TYPE ST_TrackStatus :
STRUCT
	MergePermIntlk : ARRAY[GC.MIN_MERGE_PERMINTLK..GC.MAX_MERGE_PERMINTLK] OF BOOL;
END_STRUCT
END_TYPE

(* stored: Version 1.1.0.1
   DUT ST_TrackStatus: Id {52c41a94-2924-04db-36ec-f1d788451b33} *)
